(* IEC 61131-3 sources: ml2plc/examples/models/structured_text (part 12) *)

    weights_10 : ARRAY[0..1023] OF REAL := [0.172283, 0.106642, 0.108959, -0.284027, 0.243504, -0.240655, 0.330290, 0.099606, 0.176575, 0.083414, -0.014107, 0.034331, 0.222611, 0.195157, -0.154334, -0.225464, 0.186035, -0.186008, -0.106780, -0.007384, -0.159919, -0.134954, -0.221273, -0.320173, 0.095152, 0.234545, 0.036031, -0.081243, 0.015814, 0.250287, -0.172573, -0.159019, -0.054852, 0.070771, 0.097319, 0.140936, 0.079104, 0.193619, 0.252842, 0.209296, 0.203463, 0.013421, 0.067315, 0.123931, -0.207473, 0.023318, 0.129070, 0.232349, 0.018314, -0.152895, 0.161436, -0.180890, -0.075345, -0.030392, 0.026012, 0.239923, -0.045713, -0.090956, -0.107965, -0.019277, 0.168286, -0.156662, -0.174443, 0.132358, -0.120104, 0.062717, -0.220424, -0.350078, -0.389978, 0.064511, 0.108245, -0.250363, -0.022927, 0.049594, 0.217537, -0.143713, -0.342983, 0.025154, -0.128299, 0.050483, 0.113215, -0.094273, -0.228708, -0.219715, -0.140770, 0.196364, -0.065978, 0.043672, -0.033951, 0.218606, -0.193511, -0.087589, 0.313039, 0.138918, -0.109015, -0.096872, -0.311106, -0.121318, 0.035914, 0.059759, -0.302655, -0.244137, 0.055151, 0.028730, -0.215611, 0.166152, -0.011719, -0.130943, 0.139650, 0.037964, -0.023233, 0.167527, 0.033501, 0.036641, 0.183043, 0.370582, 0.040122, -0.089372, -0.151023, 0.097306, -0.026055, 0.104931, -0.246279, -0.134042, -0.079827, 0.039389, -0.333077, 0.231532, 0.457648, -0.007698, -0.172453, 0.273185, 0.429531, -0.312808, 0.097939, 0.189175, -0.064305, 0.088152, -0.169754, 0.084893, -0.007002, -0.068024, -0.081431, -0.229271, -0.189259, -0.289942, 0.376561, -0.045270, -0.241931, -0.208321, 0.332883, -0.078408, -0.084936, 0.267926, 0.213002, 0.165506, -0.003479, -0.252180, 0.510587, -0.316997, -0.092731, -0.058917, -0.272983, 0.222480, 0.064053, 0.119469, 0.138730, -0.243328, -0.137849, 0.093328, 0.215704, 0.251980, -0.270667, -0.313309, -0.165505, -0.208583, 0.253520, -0.153595, 0.197652, 0.115504, 0.291619, -0.188014, -0.120930, -0.293720, 0.181385, -0.162253, -0.109629, -0.153464, 0.059225, 0.249463, 0.216919, 0.040383, 0.141863, 0.060170, 0.111299, 0.169653, -0.390271, 0.183970, -0.222382, -0.087671, 0.076023, 0.276760, 0.116343, 0.005845, 0.097035, -0.139421, -0.179932, -0.038168, 0.121093, 0.013039, -0.125589, 0.184791, 0.232762, 0.247056, 0.232178, 0.037920, -0.018088, -0.050510, -0.031279, -0.154764, 0.150979, -0.295636, -0.285764, 0.225964, 0.034962, 0.201042, -0.137626, 0.261234, 0.305976, -0.044416, -0.079470, -0.086079, 0.164631, 0.061417, -0.078906, 0.115023, 0.076331, 0.003390, 0.327308, 0.080462, -0.064636, -0.063342, 0.088313, -0.186020, -0.224108, -0.227707, 0.019331, 0.182962, 0.301846, 0.076243, 0.086758, 0.171452, -0.014916, -0.261342, 0.322599, 0.107263, -0.308613, 0.233097, -0.143457, -0.240650, -0.340339, 0.193940, -0.268466, -0.185200, -0.033125, 0.060978, 0.239178, -0.221807, -0.286866, 0.061810, 0.192167, -0.139503, -0.139039, 0.186929, -0.082003, 0.318103, 0.304099, 0.095908, -0.225212, -0.115199, 0.213522, -0.070028, -0.328659, -0.123167, 0.290967, 0.054711, 0.135920, 0.148910, 0.035728, -0.151008, 0.266770, -0.375333, 0.014323, -0.019379, 0.227535, -0.165065, 0.258826, -0.012944, 0.120805, -0.018290, 0.008737, -0.182124, -0.123858, 0.002958, 0.247380, -0.174737, -0.185550, 0.327737, 0.012215, 0.142727, 0.162500, -0.027943, 0.022418, -0.140562, 0.223949, -0.139202, -0.000398, -0.058497, -0.345236, -0.023818, 0.055927, -0.213166, 0.267019, 0.109094, -0.107216, -0.327065, 0.280204, 0.026999, 0.062263, -0.094313, -0.163012, 0.159902, -0.077375, -0.213250, -0.221982, -0.007775, -0.140823, -0.308292, -0.087179, -0.092401, 0.317593, 0.109718, 0.178846, -0.278912, 0.141143, 0.105545, -0.139293, 0.214422, 0.029108, 0.168299, -0.244130, 0.123023, 0.158603, 0.195359, -0.065980, 0.100870, -0.246465, 0.193647, -0.014888, 0.050222, -0.224706, 0.134822, -0.071695, -0.311419, 0.164834, 0.036925, 0.235025, 0.245503, -0.154145, -0.073790, -0.306463, -0.128804, -0.165756, 0.161038, -0.308659, -0.307926, -0.000002, 0.157067, -0.323464, -0.219380, 0.081870, -0.145446, -0.187833, 0.158573, 0.213982, 0.289394, -0.041134, -0.257900, 0.240128, 0.240368, 0.175471, 0.247867, -0.229542, 0.208854, -0.004075, -0.198774, -0.079192, 0.024001, -0.192908, 0.009208, 0.046082, 0.256710, -0.051816, 0.162976, -0.156469, 0.067293, -0.232410, -0.165859, 0.203637, 0.050521, -0.132797, 0.190456, -0.133901, 0.241903, 0.186551, 0.006898, 0.080200, -0.301116, -0.088467, -0.149174, -0.002251, -0.124423, -0.201203, 0.075967, 0.170412, -0.201278, 0.278189, -0.076042, 0.248909, -0.337676, -0.160245, 0.110007, 0.430756, 0.042573, -0.067087, -0.009378, 0.103400, -0.230516, -0.231003, 0.258105, -0.199001, 0.291249, -0.083923, -0.024625, 0.044665, -0.209391, -0.256194, 0.241611, -0.061714, 0.102455, -0.108664, -0.117878, -0.242707, 0.233309, 0.130072, -0.179273, -0.012250, -0.116236, 0.333633, -0.207854, -0.178902, 0.245079, 0.163497, -0.162975, 0.022970, -0.114253, -0.283924, -0.141254, -0.038854, 0.050053, -0.219785, 0.028346, -0.003731, 0.106553, 0.182162, -0.115632, 0.272353, -0.097840, 0.069750, -0.113570, -0.025034, 0.318486, 0.286240, 0.180103, 0.166572, 0.105172, 0.276177, 0.197487, -0.158841, 0.066383, -0.246616, 0.233556, -0.260898, 0.237399, 0.062368, 0.290960, -0.238680, -0.086516, 0.013290, 0.321653, 0.289628, 0.070572, -0.311631, 0.122021, -0.043916, -0.201292, -0.045389, -0.219363, 0.050340, 0.016358, -0.011495, -0.013630, -0.200721, 0.038771, 0.212808, -0.376513, -0.075575, -0.138494, 0.261429, 0.210696, 0.161993, -0.091646, -0.069257, -0.013123, -0.014579, -0.150370, 0.011210, 0.037860, 0.268542, 0.214858, -0.158743, 0.099199, 0.106617, -0.119096, -0.217047, -0.281159, -0.013561, -0.040896, 0.007374, -0.305835, -0.021127, -0.332499, -0.275903, 0.019077, 0.052960, -0.277409, 0.292679, -0.157464, 0.000360, 0.089573, -0.017952, -0.203217, -0.117757, -0.155011, 0.265039, 0.049836, 0.022233, 0.120586, -0.199360, -0.017568, -0.166317, 0.170938, 0.165457, 0.045632, -0.249775, -0.298162, -0.083598, 0.154531, 0.238909, -0.171492, -0.257797, 0.243346, 0.234416, 0.130320, 0.168990, -0.193712, 0.049215, -0.220860, -0.034224, -0.342114, -0.091794, -0.284842, 0.038637, -0.051852, -0.181187, -0.020978, 0.164407, -0.289722, 0.167159, -0.094716, 0.315221, 0.102350, 0.109346, -0.179846, -0.246869, -0.188476, 0.239225, -0.076139, -0.093190, -0.250823, -0.064168, -0.085364, -0.002311, 0.077880, -0.055207, 0.026922, -0.096083, -0.285327, 0.214794, 0.023161, 0.059751, -0.263913, 0.205638, 0.043162, -0.156793, -0.290027, 0.024749, -0.250236, 0.150049, 0.268845, -0.233773, 0.146997, -0.066128, -0.022977, -0.140191, -0.051843, 0.208272, 0.233819, -0.122088, -0.016243, -0.163851, 0.138372, 0.198944, 0.079420, -0.241284, -0.302888, 0.244486, 0.128862, -0.208228, 0.230048, -0.075190, -0.231913, -0.032369, -0.261644, 0.092447, -0.315003, 0.114896, 0.129825, 0.122875, 0.301763, -0.030075, -0.018081, -0.029253, -0.320159, -0.188035, 0.143382, -0.186437, -0.017232, -0.052286, 0.110700, 0.139549, 0.201258, -0.194865, -0.043933, 0.180329, 0.267740, -0.238728, 0.069253, -0.148217, -0.282364, 0.007650, -0.216262, -0.089401, 0.188749, 0.160887, 0.249590, -0.187786, 0.229560, -0.139666, -0.320477, -0.247878, 0.162484, 0.313335, -0.020400, -0.026603, -0.214849, 0.251003, -0.012518, 0.414424, 0.017157, -0.239144, 0.468889, -0.090041, 0.239761, 0.209648, 0.165673, -0.210981, -0.091000, -0.327549, 0.016095, 0.280822, 0.217226, 0.069503, -0.147461, -0.106982, -0.340036, -0.014252, -0.410382, -0.350077, -0.212908, -0.100349, -0.244298, -0.065551, -0.099630, 0.175644, -0.046378, -0.185168, -0.167246, -0.050774, -0.049952, 0.053467, 0.059175, -0.210074, -0.103228, -0.219299, 0.144060, 0.279926, -0.048009, 0.118269, 0.053479, -0.067293, 0.026087, 0.050982, -0.318531, -0.358419, -0.010575, 0.019386, -0.249029, -0.048142, 0.023493, -0.165428, 0.123698, -0.140887, -0.210041, 0.039395, 0.170219, 0.192651, 0.248423, -0.342721, -0.135088, 0.241182, -0.205243, -0.180670, 0.104035, 0.118998, -0.156160, -0.021245, -0.152837, 0.267816, -0.195864, 0.233796, 0.031097, -0.109789, -0.092834, 0.292409, -0.215144, 0.130280, 0.217063, 0.000160, 0.106179, 0.006333, 0.270528, -0.237352, -0.261159, 0.040923, 0.202982, -0.093602, 0.079623, 0.234117, 0.082825, -0.240834, -0.146769, 0.121916, 0.060845, -0.271542, 0.099722, 0.162180, 0.107957, -0.269008, 0.110029, -0.208757, 0.143843, -0.276616, 0.217388, 0.074753, -0.125457, 0.122351, -0.104234, -0.074676, 0.265085, 0.282733, 0.029273, 0.254677, 0.051715, -0.026652, 0.015909, -0.074916, -0.133114, 0.280867, -0.234281, 0.059580, 0.025924, -0.215093, -0.320628, -0.080196, 0.259291, -0.074472, 0.130335, -0.084948, -0.143250, -0.257319, -0.327923, -0.151198, -0.139865, 0.102463, -0.165763, -0.158912, -0.313267, -0.227442, 0.109861, 0.030731, -0.286002, -0.063457, -0.193754, 0.245133, 0.152417, -0.127067, 0.237635, -0.004186, -0.227178, -0.253700, -0.048737, -0.139661, 0.225958, -0.226061, 0.081229, -0.080109, 0.313959, 0.132431, 0.108710, 0.220606, 0.172431, 0.096646, -0.051313, -0.159389, 0.260342, -0.260816, 0.267087, -0.155584, -0.050812, 0.278598, 0.034435, -0.108396, 0.036017, -0.096080, 0.038691, 0.234844, -0.238547, -0.199898, -0.093337, 0.124858, -0.099312, -0.071805, -0.065751, -0.241119, -0.020975, 0.031839, 0.120518, 0.027488, 0.027341, 0.280418, 0.009611, -0.082639, -0.203516, -0.218264, 0.217235, -0.069218, -0.014592, -0.267595, 0.101731, -0.282562, -0.284809, 0.280392, -0.174080, -0.445296, -0.059798, -0.025358, 0.356295, -0.231539, 0.426815, 0.376868, 0.266828, 0.278467, -0.119267, 0.040445, -0.126245, -0.104797, -0.185307, 0.193825, -0.079105, -0.082023, 0.076038, -0.050586, 0.002755, 0.310077, -0.085438, 0.172520, 0.163448, -0.261705, -0.073560, -0.246030, -0.128170, 0.456553, -0.148266, 0.061398, -0.306320, 0.540595, 0.005749, 0.192716, -0.302604, -0.070951, 0.223005, -0.217213, -0.041680, 0.054907, 0.064077, -0.107409, 0.197957, -0.129408, -0.210510, -0.306274, -0.267641, 0.363957, 0.208692, -0.004296, 0.234353, 0.060549, -0.017092, 0.273903, 0.032570, 0.213331, -0.137710, -0.031065, 0.056870, 0.012450, -0.017812, -0.245736, 0.007675, -0.313263, -0.033795, 0.326802, -0.010816, -0.201537, 0.362160, 0.317577, -0.011858, -0.183345, 0.033902, -0.040597, 0.168911, 0.227694, 0.015293, 0.184600, 0.216630, 0.085063, 0.146565, -0.149555, -0.315725, 0.206602, 0.143192, -0.037927, -0.289462, -0.224753, 0.112222, 0.279726, -0.054142, 0.155828, -0.279028, 0.129897, -0.242403, 0.307012, -0.017188, 0.051786, -0.199068, -0.161380, -0.020222, -0.328963, -0.151638, 0.312899, 0.133312, -0.025243, -0.006013, 0.135869, -0.140045, 0.074235, 0.177620, -0.017481, -0.230667, -0.085534, -0.214468, 0.151042, -0.192704, 0.261614, 0.187512, 0.040861, -0.136434, -0.091151, 0.041760, 0.139250, 0.053344, 0.134126, 0.207952, -0.232401, 0.195006];
    bias_10 : ARRAY[0..31] OF REAL := [0.078099, 0.157173, -0.159765, 0.314937, 0.406752, -0.067901, -0.188596, -0.076708, -0.056676, 0.003795, -0.006705, -0.053043, 0.439645, -0.063894, -0.050114, -0.233493, 0.123140, 0.238549, 0.365225, -0.000873, -0.227752, 0.195915, -0.055699, -0.075604, -0.178871, -0.151893, 0.231456, -0.009470, -0.223721, -0.009080, 0.588799, -0.028734];

    weights_11 : ARRAY[0..95] OF REAL := [0.278684, -0.269775, 0.069237, 0.515927, -0.298078, 0.075745, -0.211739, -0.043259, 0.377397, 0.169311, -0.042466, -0.026853, 0.464308, -0.473260, -0.464966, -0.205327, 0.269374, -0.311708, 0.226866, 0.257922, 0.435072, 0.108650, -0.051075, -0.329926, -0.378570, 0.027921, -0.001424, -0.196133, 0.167704, 0.223128, -0.422251, -0.021511, 0.159659, -0.088594, 0.205941, -0.261449, 0.136859, -0.027370, -0.248074, -0.072602, 0.248026, 0.059923, -0.286067, 0.190599, 0.289930, -0.013859, -0.112612, 0.352590, -0.324653, 0.207672, 0.322979, 0.120654, 0.178546, 0.076933, 0.465780, 0.053887, -0.188732, -0.254513, 0.266443, 0.332247, 0.347548, 0.312686, 0.440762, 0.272259, 0.330236, 0.338985, 0.165195, 0.093332, 0.144166, 0.351201, 0.316800, 0.136666, 0.143254, -0.128643, 0.245164, -0.139607, -0.028302, 0.285889, 0.448907, -0.405661, -0.155781, 0.086899, 0.242518, 0.098446, -0.016231, -0.071013, 0.169409, -0.319740, 0.366194, -0.331713, 0.689184, -0.083837, -0.575190, -0.017942, -0.024660, -0.027264];
    bias_11 : ARRAY[0..2] OF REAL := [0.147691, 0.228653, -0.339180];

END_VAR

VAR
    (* Buffer allocation variables *)
    buffer_0 : ARRAY[0..31] OF REAL;
    buffer_1 : ARRAY[0..31] OF REAL;

    (* Temporary computation variables *)
    i : DINT;
    j : DINT;
    sum : REAL;
    max_val : REAL;
    exp_sum : REAL;

END_VAR

(* Layer 0: Fused Linear + RELU *)
FOR j := 0 TO 31 DO
    sum := 0.0;
    FOR i := 0 TO 4 DO
        sum := sum + input_data[i] * weights_0[i * 32 + j];
    END_FOR;
    buffer_1[j] := MAX(sum + bias_0[j], 0.0);
END_FOR;

(* Layer 1: Fused Linear + RELU *)
FOR j := 0 TO 31 DO
    sum := 0.0;
    FOR i := 0 TO 31 DO
        sum := sum + buffer_1[i] * weights_1[i * 32 + j];
    END_FOR;
    buffer_0[j] := MAX(sum + bias_1[j], 0.0);
END_FOR;

(* Layer 2: Fused Linear + RELU *)
FOR j := 0 TO 31 DO
    sum := 0.0;
    FOR i := 0 TO 31 DO
        sum := sum + buffer_0[i] * weights_2[i * 32 + j];
    END_FOR;
    buffer_1[j] := MAX(sum + bias_2[j], 0.0);
END_FOR;

(* Layer 3: Fused Linear + RELU *)
FOR j := 0 TO 31 DO
    sum := 0.0;
    FOR i := 0 TO 31 DO
        sum := sum + buffer_1[i] * weights_3[i * 32 + j];
    END_FOR;
    buffer_0[j] := MAX(sum + bias_3[j], 0.0);
END_FOR;

(* Layer 4: Fused Linear + RELU *)
FOR j := 0 TO 31 DO
    sum := 0.0;
    FOR i := 0 TO 31 DO
        sum := sum + buffer_0[i] * weights_4[i * 32 + j];
    END_FOR;
    buffer_1[j] := MAX(sum + bias_4[j], 0.0);
END_FOR;

(* Layer 5: Fused Linear + RELU *)
FOR j := 0 TO 31 DO
    sum := 0.0;
    FOR i := 0 TO 31 DO
        sum := sum + buffer_1[i] * weights_5[i * 32 + j];
    END_FOR;
    buffer_0[j] := MAX(sum + bias_5[j], 0.0);
END_FOR;

(* Layer 6: Fused Linear + RELU *)
FOR j := 0 TO 31 DO
    sum := 0.0;
    FOR i := 0 TO 31 DO
        sum := sum + buffer_0[i] * weights_6[i * 32 + j];
    END_FOR;
    buffer_1[j] := MAX(sum + bias_6[j], 0.0);
END_FOR;

(* Layer 7: Fused Linear + RELU *)
FOR j := 0 TO 31 DO
    sum := 0.0;
    FOR i := 0 TO 31 DO
        sum := sum + buffer_1[i] * weights_7[i * 32 + j];
    END_FOR;
    buffer_0[j] := MAX(sum + bias_7[j], 0.0);
END_FOR;

(* Layer 8: Fused Linear + RELU *)
FOR j := 0 TO 31 DO
    sum := 0.0;
    FOR i := 0 TO 31 DO
        sum := sum + buffer_0[i] * weights_8[i * 32 + j];
    END_FOR;
    buffer_1[j] := MAX(sum + bias_8[j], 0.0);
END_FOR;

(* Layer 9: Fused Linear + RELU *)
FOR j := 0 TO 31 DO
    sum := 0.0;
    FOR i := 0 TO 31 DO
        sum := sum + buffer_1[i] * weights_9[i * 32 + j];
    END_FOR;
    buffer_0[j] := MAX(sum + bias_9[j], 0.0);
END_FOR;

(* Layer 10: Fused Linear + RELU *)
FOR j := 0 TO 31 DO
    sum := 0.0;
    FOR i := 0 TO 31 DO
        sum := sum + buffer_0[i] * weights_10[i * 32 + j];
    END_FOR;
    buffer_1[j] := MAX(sum + bias_10[j], 0.0);
END_FOR;

(* Layer 11: Fused Linear + SOFTMAX *)
FOR j := 0 TO 2 DO
    sum := 0.0;
    FOR i := 0 TO 31 DO
        sum := sum + buffer_1[i] * weights_11[i * 3 + j];
    END_FOR;
    output_data[j] := sum + bias_11[j];
END_FOR;

max_val := output_data[0];
FOR i := 1 TO 2 DO
    IF output_data[i] > max_val THEN
        max_val := output_data[i];
    END_IF;
END_FOR;

exp_sum := 0.0;
FOR i := 0 TO 2 DO
    output_data[i] := EXP(output_data[i] - max_val);
    exp_sum := exp_sum + output_data[i];
END_FOR;

FOR i := 0 TO 2 DO
    output_data[i] := output_data[i] / exp_sum;
END_FOR;

END_FUNCTION_BLOCK

(* ---- test.st ---- *)
PROGRAM HelloWorld
  VAR
    OutputReg AT %MD100 : REAL;
    Counter AT %MD104 : REAL;
  END_VAR

  Counter := Counter + 1.0;
  OutputReg := Counter;
END_PROGRAM

CONFIGURATION Config0
  RESOURCE Res0 ON PLC
    TASK task0(INTERVAL := T#20ms,PRIORITY := 0);
    PROGRAM instance0 WITH task0 : HelloWorld;
  END_RESOURCE
END_CONFIGURATION
